// TwinCAT 3 PLC project FirstPLC
// ProgramVersion: 3.1.4024.0
// libraries:
//   Tc2_Standard, * (Beckhoff Automation GmbH)
//   Tc2_System, * (Beckhoff Automation GmbH)
//   Tc3_Module, * (Beckhoff Automation GmbH)
//   TcUnit, * (www.tcunit.org)
// project tree:
//   / PlcTask.TcTTO (not stored), PlcTask2.TcTTO (not stored)
//   POUs/ FB_TestSuite1.TcPOU, MAIN.TcPOU, PRG_TESTS.TcPOU, THROW_EXCEPTION.TcPOU

// ---- POUs/FB_TestSuite1.TcPOU
FUNCTION_BLOCK FB_TestSuite1 EXTENDS FB_TestSuite
VAR_INPUT
END_VAR
VAR_OUTPUT
END_VAR
VAR
END_VAR

TestCaseLongRunning();

METHOD TestCaseLongRunning
VAR_INPUT
END_VAR
TEST('TestCaseLongRunning');

// Test never finishes
//AssertTrue(2+2=4, 'Condition is not true');
//TEST_FINISHED();
END_METHOD

END_FUNCTION_BLOCK

// ---- POUs/MAIN.TcPOU
PROGRAM MAIN
VAR
	Delay : TON;
END_VAR

// Delay exception to ensure XAR run mode - do not throw in first PLC cycle
Delay(IN:= TRUE, PT:= T#5S, Q=> , ET=> );

IF Delay.Q THEN
	THROW_EXCEPTION();
END_IF

END_PROGRAM

// ---- POUs/THROW_EXCEPTION.TcPOU
FUNCTION THROW_EXCEPTION : BOOL
VAR_INPUT
END_VAR
VAR
	Value	: USINT := 100;
	Divisor	: USINT := 0;
END_VAR

Value := Value / Divisor;

END_FUNCTION

// ---- POUs/PRG_TESTS.TcPOU
PROGRAM PRG_TESTS
VAR
    fbTestSuite1Instance1 : FB_TestSuite1;
END_VAR

TcUnit.RUN();

END_PROGRAM
